// Simple logger for logging errors to specified file path on disk.
{attribute 'no_assign'}
{attribute 'enable_dynamic_creation'}
{attribute 'no_explicit_call' := 'direct call for this function block is not allowed'}
FUNCTION_BLOCK FB_DiskErrorLogger IMPLEMENTS I_ErrorLogger
VAR
	_FilePath 		: T_DiskLoggerPath;
	_Handle 		: SysTypes.RTS_IEC_HANDLE := SysTypes.RTS_INVALID_HANDLE;
	_bAutoFlush		: BOOL 			:= TRUE;
	_sDelimiter 	: STRING(1) 	:= ',';
	_sTextQualifier : STRING(1) 	:= '"';
	_sLineEnding 	: STRING(10) 	:= '$R$N';
END_VAR

// Flush the file cache automatically after logging?
// [default] TRUE - Flush after every write.
// [get] Returns the state of the auto-flush config.
// [set] Set the state of the auto-flush config.
PROPERTY AutoFlush : BOOL
GET
AutoFlush := THIS^._bAutoFlush;
END_GET
SET
THIS^._bAutoFlush := AutoFlush;
END_SET
END_PROPERTY

// Closes current log file.
METHOD Close
VAR_OUTPUT
	bIsBusy 	: BOOL;				// Is the operation still executing?
	Error 		: T_Error;			// Error produced by operation.
END_VAR
VAR
	eResult 	: E_CodesysCmpError;
END_VAR
Error := F_CreateError(	GVL_ErrorDescriptors.fbCodesysCmpErrors,
						SysFile.SysFileClose(THIS^._Handle));
END_METHOD

// Creates log entry.
METHOD PROTECTED CreateLogEntry : __XWORD // Size of message.
VAR_IN_OUT
	LoggedErrorMessage 	: T_ErrorMessage; // String to store message.
END_VAR
VAR_INPUT
	ipError				: I_Error;
END_VAR
VAR
	sDate, 
	sTimeOfDay,
	sErrorCode 			: STRING(24);
	ErrorMessage		: T_ErrorMessage;
	nCursor, nIndex 	: __UXINT;
END_VAR
IF ipError = 0 OR SIZEOF(T_ErrorMessage) < 2 THEN RETURN; END_IF

// Convert Date, time of day and error code to string.
sDate 		:= TO_STRING(ipError.Timestamp.GetDate());
sTimeOfDay 	:= TO_STRING(ipError.Timestamp.GetTimeOfDay());
sErrorCode	:= TO_STRING(ipError.Code);

// Append timestamp start text qualifier.
LoggedErrorMessage := THIS^._sTextQualifier;

// Append date.
nIndex := 0;
WHILE sDate[2 + nIndex] <> 0 DO
	nCursor := nCursor + 1;
	LoggedErrorMessage[MIN(nCursor, SIZEOF(T_ErrorMessage))] := sDate[2 + nIndex];
	nIndex := nIndex + 1;
	END_WHILE

// Append space bar.
nCursor := nCursor + 1;
LoggedErrorMessage[MIN(nCursor, SIZEOF(T_ErrorMessage))] := 32;

// Append time of day.
nIndex := 0;
WHILE sTimeOfDay[4 + nIndex] <> 0 DO
	nCursor := nCursor + 1;
	LoggedErrorMessage[MIN(nCursor, SIZEOF(T_ErrorMessage))] := sTimeOfDay[4 + nIndex];
	nIndex := nIndex + 1;
	END_WHILE
	
// Append timestamp end text qualifier.
LoggedErrorMessage[MIN(nCursor, SIZEOF(T_ErrorMessage))] := THIS^._sTextQualifier[0];

// Append delimiter.
nCursor := nCursor + 1;
LoggedErrorMessage[MIN(nCursor, SIZEOF(T_ErrorMessage))] := THIS^._sDelimiter[0];

// Append error code start text qualifier.
nCursor := nCursor + 1;
LoggedErrorMessage[MIN(nCursor, SIZEOF(T_ErrorMessage))] := THIS^._sTextQualifier[0];

// Append error code.
nIndex := 0;
WHILE sErrorCode[nIndex] <> 0 DO
	nCursor := nCursor + 1;
	LoggedErrorMessage[MIN(nCursor, SIZEOF(T_ErrorMessage))] := sErrorCode[nIndex];
	nIndex := nIndex + 1;
	END_WHILE
	
// Append error code end text qualifier.
nCursor := nCursor + 1;
LoggedErrorMessage[MIN(nCursor, SIZEOF(T_ErrorMessage))] := THIS^._sTextQualifier[0];

// Append delimiter.
nCursor := nCursor + 1;
LoggedErrorMessage[MIN(nCursor, SIZEOF(T_ErrorMessage))] := THIS^._sDelimiter[0];

// Append error code start text qualifier.
nCursor := nCursor + 1;
LoggedErrorMessage[MIN(nCursor, SIZEOF(T_ErrorMessage))] := THIS^._sTextQualifier[0];

// Append error message.
ErrorMessage := ipError.Message;
nIndex := 0;
WHILE ErrorMessage[nIndex] <> 0 DO
	nCursor := nCursor + 1;
	LoggedErrorMessage[MIN(nCursor, SIZEOF(T_ErrorMessage))] := ErrorMessage[nIndex];
	nIndex := nIndex + 1;
	END_WHILE

// Append error code end text qualifier.
nCursor := nCursor + 1;
LoggedErrorMessage[MIN(nCursor, SIZEOF(T_ErrorMessage))] := THIS^._sTextQualifier[0];

// Append line ending.
nIndex := 0;
WHILE THIS^._sLineEnding[nIndex] <> 0 DO
	nCursor := nCursor + 1;
	LoggedErrorMessage[MIN(nCursor, SIZEOF(T_ErrorMessage))] := THIS^._sLineEnding[nIndex];
	nIndex := nIndex + 1;
	END_WHILE

// Terminate string.
nCursor := nCursor + 1;
LoggedErrorMessage[MIN(nCursor, SIZEOF(T_ErrorMessage))] := 0;

// Return size of string.
CreateLogEntry := SEL(nCursor <> 0, 0, nCursor - 1);
END_METHOD

// The character used to separate logger entry fields.
// [default] ','.
// [get] Returns the delimter.
// [set] Sets the delimiter.
PROPERTY Delimiter : STRING(1)
GET
Delimiter := THIS^._sDelimiter;
END_GET
SET
THIS^._sDelimiter := Delimiter;
END_SET
END_PROPERTY

{attribute 'hide'}
METHOD FB_exit : BOOL
VAR_INPUT
	bInCopyCode : BOOL; // if TRUE, the exit method is called for exiting an instance that is copied afterwards (online change).
END_VAR
THIS^.Close();
END_METHOD

{attribute 'hide'}
METHOD FB_init : BOOL
VAR_INPUT
	bInitRetains 	: BOOL; 	// if TRUE, the retain variables are initialized (warm start / cold start)
	bInCopyCode 	: BOOL;  	// if TRUE, the instance afterwards gets moved into the copy code (online change)
	FilePath		: T_DiskLoggerPath;
END_VAR
THIS^._FilePath := FilePath;
END_METHOD

// Flushes the file cache.
METHOD Flush : I_ErrorLogger // Reference to the current instance of error logger.
VAR_OUTPUT
	bIsBusy 	: BOOL;				// Is the operation still executing?
	Error 		: T_Error;			// Error produced by operation.
END_VAR
VAR
	eResult 	: E_CodesysCmpError;
END_VAR
Flush := THIS^;

IF NOT THIS^.IsOpen THEN RETURN; END_IF

eResult := SysFile.SysFileFlush(THIS^._Handle);

IF eResult = E_CodesysCmpError.ERR_OK THEN RETURN; end_if

Error := F_CreateError(GVL_ErrorDescriptors.fbCodesysCmpErrors, eResult);
END_METHOD

// Logs the provided error message.
METHOD Invoke
VAR_INPUT
	ipError : I_Error;	 // The error message to be logged.
END_VAR
VAR_OUTPUT
	bIsBusy : BOOL;		// Is the operation still executing?
	Error 	: T_Error;	// Error produced by operation.
END_VAR
VAR
	LoggedErrorMessage 	: T_MaxString;
	nBytesWritten 		: __XWORD;
	eResult 			: E_CodesysCmpError;
END_VAR
IF ipError = 0 THEN
	Error := F_CreateError(
		GVL_ErrorDescriptors.fbCodesysCmpErrors,
		E_CodesysCmpError.ERR_INVALID_INTERFACE);
	RETURN;
	END_IF

// Open file if it's not open.
IF NOT THIS^.IsOpen THEN 
	THIS^.Open(bIsBusy => bIsBusy, Error => Error);
	IF Error.IsRaised OR bIsBusy THEN RETURN; END_IF 
	END_IF

// Write to disk.
nBytesWritten := SysFile.SysFileWrite(
	THIS^._Handle, ADR(LoggedErrorMessage),
	THIS^.CreateLogEntry(LoggedErrorMessage, ipError), ADR(eResult));

// Check for errors.
IF eResult <> E_CodesysCmpError.ERR_OK THEN 
	Error := F_CreateError(GVL_ErrorDescriptors.fbCodesysCmpErrors, eResult);
	END_IF
	
// Check if writter is busy.
bIsBusy := Error.IsNotRaised AND nBytesWritten = 0;

// Flush if not busy and auto-flush is enabled.
IF NOT bIsBusy AND Error.IsNotRaised AND THIS^._bAutoFlush THEN 
	eResult := SysFile.SysFileFlush(THIS^._Handle);
	IF eResult <> E_CodesysCmpError.ERR_OK THEN 
		Error := F_CreateError(GVL_ErrorDescriptors.fbCodesysCmpErrors, eResult);
		END_IF
	END_IF
END_METHOD

// Boolean flag indicating whether log file path is open.
// [get] Returns TRUE if the file has been openned, FALSE otherwise.
PROPERTY IsOpen : BOOL
GET
IsOpen := THIS^._Handle <> SysTypes.RTS_INVALID_HANDLE;
END_GET
END_PROPERTY

// The string used to terminate the error log entry.
// [default] '$R$N'.
// [get] Returns the line-ending.
// [set] Sets the line-ending.
PROPERTY LineEnding : STRING(1)
GET
LineEnding := THIS^._sLineEnding;
END_GET
SET
THIS^._sLineEnding := LineEnding;
END_SET
END_PROPERTY

// Opens logger file, creates it if it doesn't exist.
METHOD Open : I_ErrorLogger // Reference to the current instance of error logger.
VAR_OUTPUT
	bIsBusy 	: BOOL;				// Is the operation still executing?
	Error 		: T_Error;			// Error produced by operation.
END_VAR
VAR
	eResult 	: E_CodesysCmpError;
END_VAR
Open := THIS^;

IF THIS^.IsOpen THEN RETURN; END_IF

THIS^._Handle := SysFile.SysFileOpen(THIS^._FilePath, SysFile.AM_APPEND_PLUS, ADR(eResult));

Error := F_CreateError(GVL_ErrorDescriptors.fbCodesysCmpErrors, eResult);

bIsBusy := Error.IsNotRaised AND THIS^._Handle = SysTypes.RTS_INVALID_HANDLE;
END_METHOD

// Sets the character used to separate logger entry fields.
// [default] ','
METHOD SetDelimiter : REFERENCE TO FB_DiskErrorLogger // Reference to the current instance of error logger.
VAR_INPUT
	sValue : STRING(1); // Delimiter character.
END_VAR
SetDelimiter REF= THIS^;

THIS^._sDelimiter := sValue;
END_METHOD

// Sets the value of the string used to terminate the error log entry.
// [default] '$R$N'.
METHOD SetLineEnding : REFERENCE TO FB_DiskErrorLogger // Reference to the current instance of error logger.
VAR_INPUT
	sValue : STRING(10); // Line ending characters.
END_VAR
SetLineEnding REF= THIS^;

THIS^._sLineEnding := sValue;
END_METHOD

// Sets the character used to enclose logger entry fields.
// [default] '"'.
METHOD SetTextQualifier : REFERENCE TO FB_DiskErrorLogger // Reference to the current instance of error logger.
VAR_INPUT
	sValue : STRING(1); // Text Qualifier character.
END_VAR
SetTextQualifier REF= THIS^;

THIS^._sTextQualifier := sValue;
END_METHOD

// The character used to enclose logger entry fields.
// [default] '"'.
// [get] Returns the text qualifier.
// [set] Set the text qualifier.
PROPERTY TextQualifier : STRING(1)
GET
TextQualifier := THIS^._sTextQualifier;
END_GET
SET
THIS^._sTextQualifier := TextQualifier;
END_SET
END_PROPERTY

END_FUNCTION_BLOCK

(* stored: Version 1.1.0.1
   POU FB_DiskErrorLogger: Id {bf07c8fb-c4b4-00c4-2dc8-81af9c5efe23}, SpecialFunc None
   Folder Internal: Id {a9a452d6-d86f-095d-1e27-6e915fe03c53}
   Property AutoFlush: Id {8584c407-b91d-0d37-3c93-3614b322d90f}
   Get Get: Id {506a1180-06d0-03bc-355a-de3ae0d6ca21}
   Set Set: Id {cc35a962-3f74-098b-3192-41807790a7f8}
   Method Close: Id {657273d4-0be7-0672-1d2a-c35219928492}
   Method CreateLogEntry: Id {a64b81cf-7222-08ce-2b93-1933ad3b8e24}
   Property Delimiter: Id {a965be14-8980-098a-0686-facdbcda5b55}
   Get Get: Id {52d0affa-4ff3-0b09-2c52-06d76979b161}
   Set Set: Id {77845af1-122f-0b84-3cfd-3c4950f1cda5}
   Method FB_exit: Id {54a3a68e-3b01-01ed-2302-97545d26a69e}
   Method FB_init: Id {c724ded2-9460-0e4b-11ab-2f4d7def4683}
   Method Flush: Id {f8b1fa13-2faf-0760-28e7-5ec2c2aed697}
   Method Invoke: Id {59e699e2-7a12-01ea-1ac7-9de854c5852e}
   Property IsOpen: Id {ad810b2d-1ad8-01c7-0b67-c9787cf786d2}
   Get Get: Id {24c369ce-8831-0ff8-0559-61f448a803f7}
   Property LineEnding: Id {8797567b-2ab6-0047-16c4-1823649a5b9f}
   Get Get: Id {c4dc78ff-af6e-03e0-18f6-774717db0796}
   Set Set: Id {ad0d6d5a-e96d-0805-047b-290fd214c47f}
   Method Open: Id {a9d72e4d-bcf0-02de-37fc-35cd2080eeee}
   Method SetDelimiter: Id {c65adf51-c44e-0bc1-1c26-85c083bc7d41}
   Method SetLineEnding: Id {63b8a44c-8194-0cb7-2482-a4c3d39edc61}
   Method SetTextQualifier: Id {a52b0548-14a2-0775-08cd-329106d33ca7}
   Property TextQualifier: Id {ee0f8a21-8469-0939-0690-bf6c7dcbe421}
   Get Get: Id {ad0af364-8771-0250-2eeb-62ee922c13c8}
   Set Set: Id {a8611ce6-9a7f-0b5f-330d-ec7bdc6a8ced} *)
